(* IEC 61131-3 sources: repolevel_ST_code_completion/output/0127完整版本_带planner/repoeval_traffic_light/readful_result_no_provide, 3 files *)

(* ---- F_SecondsToTime.st ---- *)
F_SecondsToTime := DWORD_TO_TIME(dwSeconds * 1000);
RETURN;
END_FUNCTION

(* ---- F_TimeToSeconds.st ---- *)
F_TimeToSeconds := DINT_TO_DWORD(TRUNC(TIME_TO_DWORD(tTime) / 1000.0));
RETURN;
END_FUNCTION

(* ---- FB_CountdownTimer.st ---- *)
VAR
	nTotalSeconds		:	UINT;	//总秒数
	nElapsedSeconds		:	UINT;	//已过秒数
END_VAR

// 将TIME转换为秒
nTotalSeconds := TO_UINT(TIME_TO_DWORD(tTotalTime) / 1000);
nElapsedSeconds := TO_UINT(TIME_TO_DWORD(tElapsedTime) / 1000);

// 检查是否已经过了总时间
IF tElapsedTime >= tTotalTime THEN
	nRemainingSeconds := 0;
ELSE
	// 计算剩余秒数
	nRemainingSeconds := nTotalSeconds - nElapsedSeconds;
END_IF;
END_FUNCTION_BLOCK
